// TIA Portal V16 export
// export: Created 2023-03-29T11:05:05.3562269Z, ExportSetting WithDefaults, DisplayName Totally Integrated Automation Portal, DisplayVersion V16 Update 6, DisplayName TIA Portal Version Control Interface, DisplayVersion V16 Update 2, DisplayName TIA Portal Openness, DisplayVersion V16 Update 6, DisplayName STEP 7 Professional, DisplayVersion V16 Update 6, DisplayName STEP 7 Safety, DisplayVersion V16, DisplayName WinCC Advanced, DisplayVersion V16 Update 6
VAR_GLOBAL   // PLC tag table "ModbusTCP"
   memTrgServer_1 AT %M106.0 : Bool;
   memTrgServer_2 AT %M106.1 : Bool;
   memTrgServer_3 AT %M106.2 : Bool;
   DISCONNECT_SERVER_1 AT %M106.3 : Bool;
   DISCONNECT_SERVER_2 AT %M106.4 : Bool;
   DISCONNECT_SERVER_3 AT %M106.5 : Bool;
   memRisingTriger_Data_4 AT %M107.1 : Bool;   // pamieć zbocza narastającego przekazania danej do wysłania
   memRisingTriger_Data_11 AT %M108.0 : Bool;   // pamieć zbocza narastającego przekazania danej do wysłania
   memRisingTriger_Data_5 AT %M107.2 : Bool;   // pamieć zbocza narastającego przekazania danej do wysłania
   memRisingTriger_Data_8 AT %M107.5 : Bool;   // pamieć zbocza narastającego przekazania danej do wysłania
   memRisingTriger_Data_1 AT %M106.6 : Bool;   // pamieć zbocza narastającego przekazania danej do wysłania
   memRisingTriger_Data_13 AT %M108.2 : Bool;   // pamieć zbocza narastającego przekazania danej do wysłania
   memRisingTriger_Data_2 AT %M106.7 : Bool;   // pamieć zbocza narastającego przekazania danej do wysłania
   memRisingTriger_Data_6 AT %M107.3 : Bool;   // pamieć zbocza narastającego przekazania danej do wysłania
   memRisingTriger_Data_10 AT %M107.7 : Bool;   // pamieć zbocza narastającego przekazania danej do wysłania
   memRisingTriger_Data_12 AT %M108.1 : Bool;   // pamieć zbocza narastającego przekazania danej do wysłania
   memRisingTriger_Data_3 AT %M107.0 : Bool;   // pamieć zbocza narastającego przekazania danej do wysłania
   memRisingTriger_Data_9 AT %M107.6 : Bool;   // pamieć zbocza narastającego przekazania danej do wysłania
   memRisingTriger_Data_7 AT %M107.4 : Bool;   // pamieć zbocza narastającego przekazania danej do wysłania
   DISCONNECT_SERVER_4 AT %M108.3 : Bool;
   memTrgServer_4 AT %M108.4 : Bool;
   memTrig_Client_Receiving_16 AT %M110.4 : Bool;
   memTrig_Client_Receiving_7 AT %M109.3 : Bool;
   memTrig_Client_Receiving_11 AT %M109.7 : Bool;
   memRisingTriger_Data_1_2 AT %M110.6 : Bool;   // pamieć zbocza narastającego przekazania danej do wysłania
   memRisingTriger_Data_1_1 AT %M110.5 : Bool;   // pamieć zbocza narastającego przekazania danej do wysłania
   memTrig_Client_Receiving_5 AT %M109.1 : Bool;
   memTrig_Client_Receiving_13 AT %M110.1 : Bool;
   memTrig_Client_Receiving_14 AT %M110.2 : Bool;
   memTrig_Client_Receiving_3 AT %M108.7 : Bool;
   memTrig_Client_Receiving_8 AT %M109.4 : Bool;
   memTrig_Client_Receiving_10 AT %M109.6 : Bool;
   memTrig_Client_Receiving_6 AT %M109.2 : Bool;
   memTrig_Client_Receiving_12 AT %M110.0 : Bool;
   memTrig_Client_Receiving_2 AT %M108.6 : Bool;
   memTrig_Client_Receiving_1 AT %M108.5 : Bool;
   memTrig_Client_Receiving_4 AT %M109.0 : Bool;
   memTrig_Client_Receiving_9 AT %M109.5 : Bool;
   memTrig_Client_Receiving_15 AT %M110.3 : Bool;
   memRisingTriger_Data_16 AT %M111.2 : Bool;
   memRisingTriger_Data_14 AT %M111.0 : Bool;
   memRisingTriger_Data_15 AT %M111.1 : Bool;
   memRisingTriger_Data_47 AT %M115.1 : Bool;
   memTrig_Client_Receiving_17 AT %M120.2 : Bool;
   memTrig_Client_Receiving_87 AT %M129.0 : Bool;
   memTrig_Client_Receiving_23 AT %M121.0 : Bool;
   memRisingTriger_Data_29 AT %M112.7 : Bool;
   memTrig_Client_Receiving_84 AT %M128.5 : Bool;
   memTrig_Client_Receiving_43 AT %M123.4 : Bool;
   memRisingTriger_Data_63 AT %M117.1 : Bool;
   memTrig_Client_Receiving_74 AT %M127.3 : Bool;
   memRisingTriger_Data_69 AT %M117.7 : Bool;
   memRisingTriger_Data_70 AT %M118.0 : Bool;
   memTrig_Client_Receiving_32 AT %M122.1 : Bool;
   memRisingTriger_Data_80 AT %M119.2 : Bool;
   memTrig_Client_Receiving_65 AT %M126.2 : Bool;
   memTrig_Client_Receiving_71 AT %M127.0 : Bool;
   memTrig_Client_Receiving_36 AT %M122.5 : Bool;
   memRisingTriger_Data_84 AT %M119.6 : Bool;
   memRisingTriger_Data_68 AT %M117.6 : Bool;
   memTrig_Client_Receiving_49 AT %M124.2 : Bool;
   memRisingTriger_Data_85 AT %M119.7 : Bool;
   memRisingTriger_Data_36 AT %M113.6 : Bool;
   memTrig_Client_Receiving_76 AT %M127.5 : Bool;
   memTrig_Client_Receiving_70 AT %M126.7 : Bool;
   memTrig_Client_Receiving_89 AT %M129.2 : Bool;
   memRisingTriger_Data_19 AT %M111.5 : Bool;
   memRisingTriger_Data_31 AT %M113.1 : Bool;
   memTrig_Client_Receiving_20 AT %M120.5 : Bool;
   memTrig_Client_Receiving_48 AT %M124.1 : Bool;
   memTrig_Client_Receiving_56 AT %M125.1 : Bool;
   memRisingTriger_Data_44 AT %M114.6 : Bool;
   memTrig_Client_Receiving_82 AT %M128.3 : Bool;
   memTrig_Client_Receiving_58 AT %M125.3 : Bool;
   memTrig_Client_Receiving_67 AT %M126.4 : Bool;
   memRisingTriger_Data_57 AT %M116.3 : Bool;
   memTrig_Client_Receiving_80 AT %M128.1 : Bool;
   memRisingTriger_Data_52 AT %M115.6 : Bool;
   memTrig_Client_Receiving_69 AT %M126.6 : Bool;
   memRisingTriger_Data_64 AT %M117.2 : Bool;
   memTrig_Client_Receiving_60 AT %M125.5 : Bool;
   memTrig_Client_Receiving_62 AT %M125.7 : Bool;
   memRisingTriger_Data_26 AT %M112.4 : Bool;
   memRisingTriger_Data_82 AT %M119.4 : Bool;
   memRisingTriger_Data_72 AT %M118.2 : Bool;
   memTrig_Client_Receiving_26 AT %M121.3 : Bool;
   memRisingTriger_Data_73 AT %M118.3 : Bool;
   memRisingTriger_Data_46 AT %M115.0 : Bool;
   memTrig_Client_Receiving_73 AT %M127.2 : Bool;
   memTrig_Client_Receiving_24 AT %M121.1 : Bool;
   memRisingTriger_Data_42 AT %M114.4 : Bool;
   memTrig_Client_Receiving_78 AT %M127.7 : Bool;
   memRisingTriger_Data_27 AT %M112.5 : Bool;
   memTrig_Client_Receiving_25 AT %M121.2 : Bool;
   memRisingTriger_Data_34 AT %M113.4 : Bool;
   memTrig_Client_Receiving_30 AT %M121.7 : Bool;
   memTrig_Client_Receiving_47 AT %M124.0 : Bool;
   memRisingTriger_Data_71 AT %M118.1 : Bool;
   memRisingTriger_Data_18 AT %M111.4 : Bool;
   memRisingTriger_Data_33 AT %M113.3 : Bool;
   memTrig_Client_Receiving_85 AT %M128.6 : Bool;
   memRisingTriger_Data_17 AT %M111.3 : Bool;
   memRisingTriger_Data_74 AT %M118.4 : Bool;
   memRisingTriger_Data_35 AT %M113.5 : Bool;
   memTrig_Client_Receiving_42 AT %M123.3 : Bool;
   memTrig_Client_Receiving_37 AT %M122.6 : Bool;
   memTrig_Client_Receiving_22 AT %M120.7 : Bool;
   memRisingTriger_Data_81 AT %M119.3 : Bool;
   memTrig_Client_Receiving_18 AT %M120.3 : Bool;
   memRisingTriger_Data_87 AT %M120.1 : Bool;
   memRisingTriger_Data_62 AT %M117.0 : Bool;
   memTrig_Client_Receiving_19 AT %M120.4 : Bool;
   memRisingTriger_Data_40 AT %M114.2 : Bool;
   memTrig_Client_Receiving_46 AT %M123.7 : Bool;
   memTrig_Client_Receiving_63 AT %M126.0 : Bool;
   memTrig_Client_Receiving_35 AT %M122.4 : Bool;
   memRisingTriger_Data_83 AT %M119.5 : Bool;
   memTrig_Client_Receiving_21 AT %M120.6 : Bool;
   memTrig_Client_Receiving_83 AT %M128.4 : Bool;
   memRisingTriger_Data_39 AT %M114.1 : Bool;
   memRisingTriger_Data_53 AT %M115.7 : Bool;
   memTrig_Client_Receiving_44 AT %M123.5 : Bool;
   memRisingTriger_Data_45 AT %M114.7 : Bool;
   memRisingTriger_Data_37 AT %M113.7 : Bool;
   memTrig_Client_Receiving_38 AT %M122.7 : Bool;
   memTrig_Client_Receiving_79 AT %M128.0 : Bool;
   memRisingTriger_Data_32 AT %M113.2 : Bool;
   memRisingTriger_Data_22 AT %M112.0 : Bool;
   memTrig_Client_Receiving_72 AT %M127.1 : Bool;
   memTrig_Client_Receiving_31 AT %M122.0 : Bool;
   memTrig_Client_Receiving_68 AT %M126.5 : Bool;
   memTrig_Client_Receiving_55 AT %M125.0 : Bool;
   memRisingTriger_Data_67 AT %M117.5 : Bool;
   memRisingTriger_Data_41 AT %M114.3 : Bool;
   memRisingTriger_Data_28 AT %M112.6 : Bool;
   memRisingTriger_Data_61 AT %M116.7 : Bool;
   memTrig_Client_Receiving_64 AT %M126.1 : Bool;
   memTrig_Client_Receiving_50 AT %M124.3 : Bool;
   memRisingTriger_Data_76 AT %M118.6 : Bool;
   memRisingTriger_Data_30 AT %M113.0 : Bool;
   memRisingTriger_Data_58 AT %M116.4 : Bool;
   memRisingTriger_Data_75 AT %M118.5 : Bool;
   memRisingTriger_Data_60 AT %M116.6 : Bool;
   memRisingTriger_Data_56 AT %M116.2 : Bool;
   memTrig_Client_Receiving_34 AT %M122.3 : Bool;
   memTrig_Client_Receiving_52 AT %M124.5 : Bool;
   memTrig_Client_Receiving_27 AT %M121.4 : Bool;
   memRisingTriger_Data_54 AT %M116.0 : Bool;
   memRisingTriger_Data_25 AT %M112.3 : Bool;
   memTrig_Client_Receiving_33 AT %M122.2 : Bool;
   memRisingTriger_Data_23 AT %M112.1 : Bool;
   memRisingTriger_Data_66 AT %M117.4 : Bool;
   memTrig_Client_Receiving_88 AT %M129.1 : Bool;
   memRisingTriger_Data_51 AT %M115.5 : Bool;
   memRisingTriger_Data_43 AT %M114.5 : Bool;
   memRisingTriger_Data_86 AT %M120.0 : Bool;
   memRisingTriger_Data_65 AT %M117.3 : Bool;
   memTrig_Client_Receiving_66 AT %M126.3 : Bool;
   memTrig_Client_Receiving_28 AT %M121.5 : Bool;
   memTrig_Client_Receiving_51 AT %M124.4 : Bool;
   memTrig_Client_Receiving_59 AT %M125.4 : Bool;
   memRisingTriger_Data_38 AT %M114.0 : Bool;
   memTrig_Client_Receiving_45 AT %M123.6 : Bool;
   memRisingTriger_Data_79 AT %M119.1 : Bool;
   memTrig_Client_Receiving_81 AT %M128.2 : Bool;
   memRisingTriger_Data_50 AT %M115.4 : Bool;
   memTrig_Client_Receiving_86 AT %M128.7 : Bool;
   memRisingTriger_Data_55 AT %M116.1 : Bool;
   memTrig_Client_Receiving_41 AT %M123.2 : Bool;
   memTrig_Client_Receiving_54 AT %M124.7 : Bool;
   memRisingTriger_Data_49 AT %M115.3 : Bool;
   memTrig_Client_Receiving_53 AT %M124.6 : Bool;
   memTrig_Client_Receiving_61 AT %M125.6 : Bool;
   memRisingTriger_Data_59 AT %M116.5 : Bool;
   memTrig_Client_Receiving_77 AT %M127.6 : Bool;
   memTrig_Client_Receiving_29 AT %M121.6 : Bool;
   memRisingTriger_Data_77 AT %M118.7 : Bool;
   memRisingTriger_Data_48 AT %M115.2 : Bool;
   memTrig_Client_Receiving_40 AT %M123.1 : Bool;
   memRisingTriger_Data_24 AT %M112.2 : Bool;
   memTrig_Client_Receiving_57 AT %M125.2 : Bool;
   memRisingTriger_Data_20 AT %M111.6 : Bool;
   timeDISCONECT_TCP_SERVER_1 AT %M111.7 : Bool;
   timeDISCONECT_TCP_SERVER_2 AT %M123.0 : Bool;
   timeDISCONECT_TCP_SERVER_3 AT %M119.0 : Bool;
   timeDISCONECT_TCP_SERVER_4 AT %M127.4 : Bool;
END_VAR
